TYPE ST_P10A_Pult_OUT :
STRUCT
	bLedHakenpos	: BOOL; // Hakenposition Anfahren; LDT-BU, 2FDI-NO, 1DO; P10A-51SJ3
	bLedRichtungL	: BOOL; // Richtung Links; LDT-WH, 1DI-NO, 1DO; P10A-21SJ1
	bLedRichtungR	: BOOL; // Richtung Rechts; LDT-WH, 1DI-NO, 1DO; P10A-21SJ2
END_STRUCT
END_TYPE

(* stored: Version 1.1.0.1
   DUT ST_P10A_Pult_OUT: Id {cee7ac8d-7b0e-4ef1-b0eb-9d7d9a5d1138} *)
